TYPE ST_12ViciValveSampleNames :
STRUCT
	{attribute 'pytmc' := '
        pv: 01
        io: io
     '}
     s1 : STRING;
     {attribute 'pytmc' := '
        pv: 02
        io: io
     '}
     s2 : STRING;
     {attribute 'pytmc' := '
        pv: 03
        io: io
     '}
     s3 : STRING;
     {attribute 'pytmc' := '
        pv: 04
        io: io
     '}
     s4 : STRING;
	       {attribute 'pytmc' := '
        pv: 05
        io: io
     '}
     s5 : STRING;
     {attribute 'pytmc' := '
        pv: 06
        io: io
     '}
     s6 : STRING;
     {attribute 'pytmc' := '
        pv: 07
        io: io
     '}
     s7 : STRING;
     {attribute 'pytmc' := '
        pv: 08
        io: io
     '}
     s8 : STRING;
	       {attribute 'pytmc' := '
        pv: 09
        io: io
     '}
     s9 : STRING;
     {attribute 'pytmc' := '
        pv: 10
        io: io
     '}
     s10 : STRING;
     {attribute 'pytmc' := '
        pv: 11
        io: io
     '}
     s11 : STRING;
     {attribute 'pytmc' := '
        pv: 12
        io: io
     '}
     s12 : STRING;
END_STRUCT
END_TYPE

(* stored: Version 1.1.0.1, ProductVersion 3.1.4024.12
   DUT ST_12ViciValveSampleNames: Id {3a13c3fd-2ef6-436c-b65e-9eb376830a93} *)
